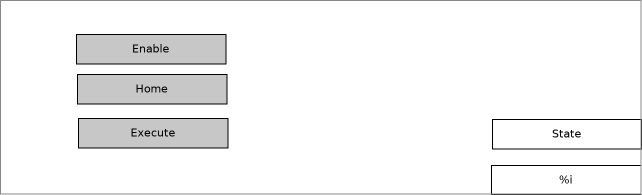
VISUALIZATION Visualization  // 642x195
    Rectangle (76,34 150x30), "Enable", colour toggle: MAIN.bEnable
        toggle MAIN.bEnable
    Rectangle (77,74 150x30), "Home", colour toggle: MAIN.homeAxi
        tap MAIN.homeAxi
    Rectangle (78,118 150x30), "Execute", colour toggle: MAIN.executeGcode
        tap MAIN.executeGcode
    Rectangle (491,165 150x30), "%i", text variable: MAIN.State
    Rectangle (492,119 150x30), "State"
END_VISUALIZATION

(* stored: Version 1.1.0.1, ProductVersion 3.1.4024.11
   Visu Visualization: Id {08d3b490-6e42-48e2-a4f5-a5f079737388} *)
